Staubli VAL3: clkBack.pgx

program clkBack()
begin
  userPage("firstpage")
end
